FUNCTION_BLOCK PickerSequenceBoot EXTENDS PickerSequence IMPLEMENTS ZCore.ISequence
VAR
  _step : ZCore.Step(PickerStep.BootBegin, PickerStep.BootEnd);
END_VAR

IF OnStart(_step) THEN
  ; // init custom sequence variables here ...
END_IF

REPEAT
  LogStep();

  CASE _step.Index OF
    (* -------------------------------------------------------------------------------------------------------------------------------- *)
    PickerStep.BootBegin:
    (* -------------------------------------------------------------------------------------------------------------------------------- *)
      IF _step.OnEntry()
      THEN
        // initialize equipment
        _io();
        _actuator();
        _fieldbus();
        _axis();
        _unit();
      END_IF
      
      _parent._objectManager.Cyclic();      
      Assert(_parent._objectManager);
      IF _parent._objectManager.Booted
      THEN
        _step.SetNext(PickerStep.BootEnd);
      END_IF

    (* -------------------------------------------------------------------------------------------------------------------------------- *)
    PickerStep.BootEnd:
    (* -------------------------------------------------------------------------------------------------------------------------------- *)
      SetBusy(FALSE);
      
  ELSE
    Abort('sequence contains unhandled step');
  END_CASE
UNTIL _step.IsNotRepeatable() OR_ELSE NOT Busy END_REPEAT

END_FUNCTION_BLOCK

(* stored: Version 1.1.0.1
   POU PickerSequenceBoot: Id {f492b112-acd4-4258-ab00-c5decb7eaad6}, SpecialFunc None *)
